TYPE (* SoftKeyActivationCode Struct *)
  (* Version 1.0, 2025-07-21, franz *)
  SoftKeyActivationCode_S : STRUCT
    code : USINT := 255;
    bCyclic : BOOL := FALSE; (* do not repeat every 200ms if this is set FALSE *)
  END_STRUCT;
END_TYPE
